(* Logix 5000 project; controller Savage_Saw vendor 1 type 14 code 152 rev 33.16; software revision 33.04 *)

TASK MainTask (continuous, watchdog 500 ms) : MainProgram

MODULES
   Local : vendor 1 type 14 code 152 (PointIO 0, rev 33.16)
      Kane : vendor 590 type 43 code 5 (Ethernet 192.168.3.12, rev 1.1, StandardDataDriven RPI 20 ms)
      HPU_Panel : 1734-AENTR (Ethernet 192.168.3.11, rev 7.13, Output RPI 20 ms)
         AnalogIn7_8 : 1734-IE2V (PointIO 2, rev 3.5, Input RPI 80 ms)
         AnalogIn5_6 : 1734-IE2V (PointIO 1, rev 3.5, Input RPI 80 ms)
         InputDC0_8 : 1734-IB8 (PointIO 3, rev 3.22)
         InputDC9_17 : 1734-IB8 (PointIO 4, rev 3.22)
         OutputDC0_3 : vendor 1 type 7 code 134 (PointIO 5, rev 3.2)
         OutputDC4_7 : vendor 1 type 7 code 134 (PointIO 6, rev 3.2)
         OutputDC8_11 : vendor 1 type 7 code 134 (PointIO 7, rev 3.2)
      Analog0_1 : 1734-IE2V (PointIO 2, rev 3.5, Input RPI 80 ms)
      Analog2_3 : 1734-IE2V (PointIO 3, rev 3.4, Input RPI 80 ms)
      Discrete_IO : Embedded (PointIO 1, rev 33.11, Output RPI 20 ms)
       : 1734-OA4 (PointIO 4, rev 3.22, Output RPI 20 ms)
       : 1734-OA4 (PointIO 5, rev 3.22, Output RPI 20 ms)
       : 1734-OA4 (PointIO 6, rev 3.22, Output RPI 20 ms)
END_MODULES

TYPE Kane_OUT_DATA1 :
STRUCT
   Unassigned_Var_Table_12 : REAL;
   Unassigned_Var_Table_13 : REAL;
   Unassigned_Var_Table_14 : REAL;
   Unassigned_Var_Table_15 : REAL;
   Unassigned_Var_Table_16 : REAL;
   Unassigned_Var_Table_17 : REAL;
   Unassigned_Var_Table_18 : REAL;
   Unassigned_Var_Table_19 : REAL;
   Unassigned_Var_Table_20 : REAL;
   Unassigned_Var_Table_21 : REAL;
END_STRUCT
END_TYPE

TYPE RMC_IN :
STRUCT
   xCutStatus : DINT;
   yBedStatus : DINT;
   zDepthStatus : DINT;
   xCutPosition : REAL;
   yBedPosition : REAL;
   zDepthPosition : REAL;
END_STRUCT
END_TYPE

TYPE RMC_OUT :
STRUCT
   xCutPosnCommand : REAL;
   yBedPosnCommand : REAL;
   zDepthPosnCommand : REAL;
   xCutVelocity : REAL;
   yBedVelocity : REAL;
   zDepthVelocity : REAL;
END_STRUCT
END_TYPE

VAR_GLOBAL   (* controller tags *)
   RMC_Busy : BOOL;
   RMC_In : RMC_IN := (xCutStatus := 67113540, yBedStatus := 67113540, zDepthStatus := 1108831372, xCutPosition := 37.856003);
   RMC_Out : RMC_OUT := (xCutPosnCommand := 9.999, yBedPosnCommand := 2.2, zDepthPosnCommand := 3.3, xCutVelocity := 4.4, yBedVelocity := 5.5, zDepthVelocity := 69.6);
   RMC_SendRequest : BOOL;
   tbOnOff : BOOL;
   test : DINT;
   tmrTest : TIMER := (PRE := 1000);
END_VAR

PROGRAM MainProgram   (* main routine RMC *)

ROUTINE RMC   (* ladder *)
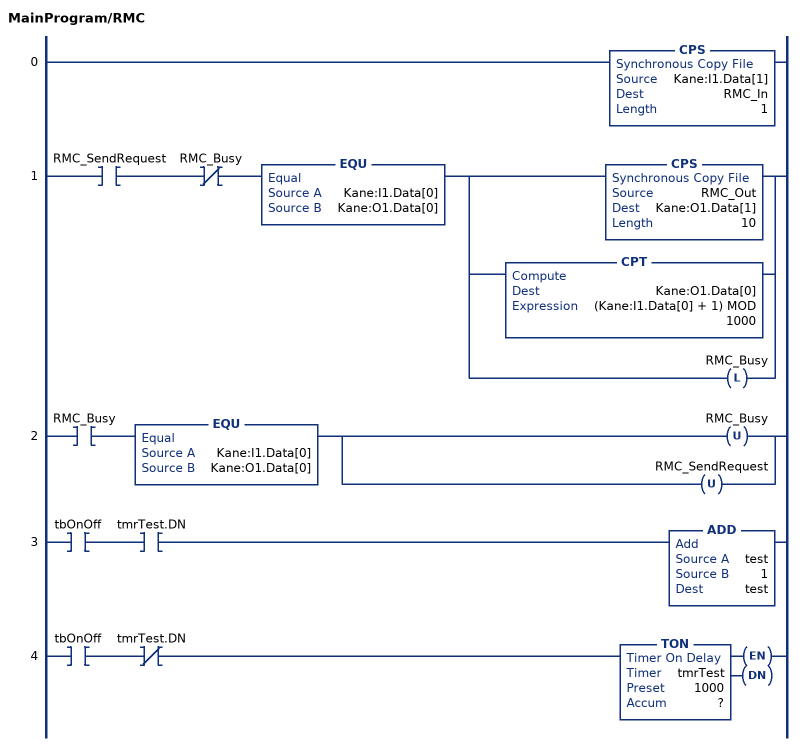
   0: CPS(Kane:I1.Data[1],RMC_In,1);
   1: XIC(RMC_SendRequest)XIO(RMC_Busy)EQU(Kane:I1.Data[0],Kane:O1.Data[0])[CPS(RMC_Out,Kane:O1.Data[1],10) ,CPT(Kane:O1.Data[0],(Kane:I1.Data[0] + 1) MOD 1000) ,OTL(RMC_Busy) ];
   2: XIC(RMC_Busy)EQU(Kane:I1.Data[0],Kane:O1.Data[0])[OTU(RMC_Busy) ,OTU(RMC_SendRequest) ];
   3: XIC(tbOnOff)XIC(tmrTest.DN)ADD(test,1,test);
   4: XIC(tbOnOff)XIO(tmrTest.DN)TON(tmrTest,?,?);
END_ROUTINE
END_PROGRAM
